FUNCTION_BLOCK SkillVcmOn (* Basic Function Block Type *)
  (* Standard: 61499-2 *)
  (* Version 0.0, 2/16/2024, midxav, Template *)
  PACKAGE Main;
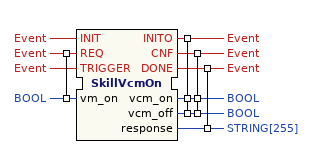
  EVENT_INPUT
    INIT; (* Initialization Request *)
    REQ WITH vm_on; (* Normal Execution Request *)
    TRIGGER;
  END_EVENT
  EVENT_OUTPUT
    INITO WITH vcm_on, vcm_off; (* Initialization Confirm *)
    CNF WITH vcm_on, vcm_off; (* Execution Confirmation *)
    DONE WITH response;
  END_EVENT
  VAR_INPUT
    vm_on : BOOL;
  END_VAR
  VAR_OUTPUT
    vcm_on : BOOL;
    vcm_off : BOOL;
    response : STRING[255];
  END_VAR
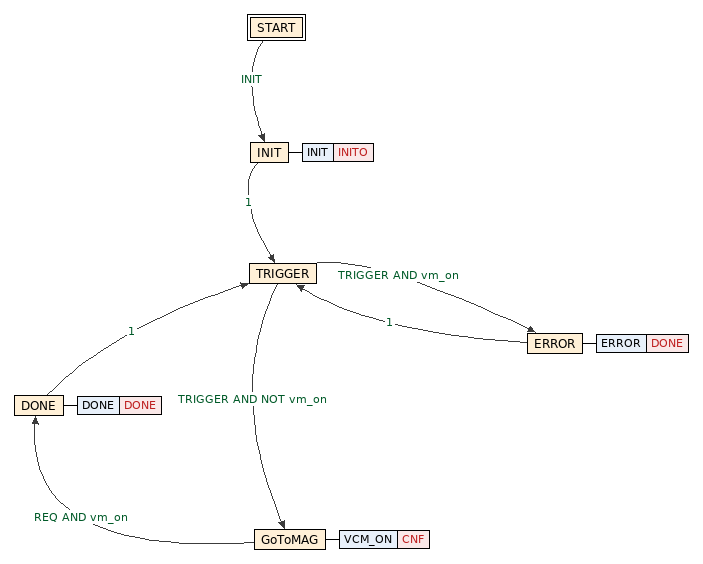
  EC_STATES
    START; (* Initial State *)
    INIT : INIT -> INITO; (* Initialization *)
    GoToMAG : VCM_ON -> CNF;
    DONE : DONE -> DONE;
    TRIGGER;
    ERROR : ERROR -> DONE;
  END_STATES
  EC_TRANSITIONS
    START TO INIT := INIT;
    TRIGGER TO GoToMAG := TRIGGER AND NOT vm_on;
    GoToMAG TO DONE := REQ AND vm_on;
    DONE TO TRIGGER := 1;
    INIT TO TRIGGER := 1;
    TRIGGER TO ERROR := TRIGGER AND vm_on;
    ERROR TO TRIGGER := 1;
  END_TRANSITIONS
  ALGORITHM INIT IN ST: (* Initialization algorithm *)
vcm_on :=FALSE;
vcm_off :=TRUE;
  END_ALGORITHM
  ALGORITHM VCM_ON IN ST:
vcm_on := TRUE;
vcm_off := FALSE;
  END_ALGORITHM
  ALGORITHM VCM_OFF IN ST:
vcm_on := FALSE;
vcm_off := TRUE;
  END_ALGORITHM
  ALGORITHM DONE IN ST:
response:='PICKED WP';
  END_ALGORITHM
  ALGORITHM ERROR IN ST:
response:='ALREADY PICK IS ON';
TRIGGER:=FALSE;
  END_ALGORITHM
END_FUNCTION_BLOCK
